// Mitsubishi GX Works2 project: BookEX6_25 Transfer   PLC: Q13UDV

// global labels: Global
VAR_GLOBAL
  bVar0 AT M5000 : BOOL;
  abArray0 AT M5010 : ARRAY [0..49] OF BOOL;
  sStr0 AT D5000 : STRING[199];
  sStr1 AT D5100 : STRING[199];
  sStr2 AT D5200 : STRING[199];
  sStr3 AT D5300 : STRING[199];
  sStr4 AT D5400 : STRING[199];
  sStr5 AT D5500 : STRING[199];
  sStr6 AT D5600 : STRING[199];
  sStr7 AT D5700 : STRING[199];
  sStr8 AT D5800 : STRING[199];
  sStr9 AT D5900 : STRING[199];
  iVar0 AT D4500 : INT;
  iVar1 AT D4501 : INT;
  iVar2 AT D4502 : INT;
  iVar3 AT D4503 : INT;
  iVar4 AT D4504 : INT;
  iVar5 AT D4505 : INT;
  iVar6 AT D4506 : INT;
  iVar7 AT D4507 : INT;
  iVar8 AT D4508 : INT;
  iVar9 AT D4509 : INT;
  dVar0 AT D4510 : DINT;
  dVar1 AT D4512 : DINT;
  dVar2 AT D4514 : DINT;
  dVar3 AT D4516 : DINT;
  dVar4 AT D4518 : DINT;
  dVar5 AT D4520 : DINT;
  dVar6 AT D4522 : DINT;
  dVar7 AT D4524 : DINT;
  dVar8 AT D4526 : DINT;
  dVar9 AT D4528 : DINT;
  wVar0 AT D4530 : WORD;
  wVar1 AT D4531 : WORD;
  wVar2 AT D4532 : WORD;
  wVar3 AT D4533 : WORD;
  wVar4 AT D4534 : WORD;
  wVar5 AT D4535 : WORD;
  wVar6 AT D4536 : WORD;
  wVar7 AT D4537 : WORD;
  wVar8 AT D4538 : WORD;
  wVar9 AT D4539 : WORD;
  dwVar0 AT D4540 : DWORD;
  dwVar1 AT D4542 : DWORD;
  dwVar2 AT D4544 : DWORD;
  dwVar3 AT D4546 : DWORD;
  dwVar4 AT D4548 : DWORD;
  dwVar5 AT D4550 : DWORD;
  dwVar6 AT D4552 : DWORD;
  dwVar7 AT D4554 : DWORD;
  dwVar8 AT D4556 : DWORD;
  dwVar9 AT D4558 : DWORD;
  fsVar0 AT D4560 : REAL;
  fsVar1 AT D4562 : REAL;
  fsVar2 AT D4564 : REAL;
  fsVar3 AT D4566 : REAL;
  fsVar4 AT D4568 : REAL;
  fsVar5 AT D4570 : REAL;
  fsVar6 AT D4572 : REAL;
  fsVar7 AT D4574 : REAL;
  fsVar8 AT D4576 : REAL;
  fsVar9 AT D4578 : REAL;
  fdVar0 AT D4580 : LREAL;
  tTime0 AT D4620 : TIME;
  tTime1 AT D4622 : TIME;
  tTime2 AT D4624 : TIME;
  tTime3 AT D4626 : TIME;
  tTime4 AT D4628 : TIME;
  tTime5 AT D4630 : TIME;
  tTime6 AT D4632 : TIME;
  tTime7 AT D4634 : TIME;
  tTime8 AT D4636 : TIME;
  tTime9 AT D4638 : TIME;
  tTime10 AT D4640 : TIME;
  bVar1 AT M5001 : BOOL;
  bVar2 AT M5002 : BOOL;
  bVar3 AT M5003 : BOOL;
  bVar4 AT M5004 : BOOL;
  bVar5 AT M5005 : BOOL;
  bVar6 AT M5006 : BOOL;
  bVar7 AT M5007 : BOOL;
  bVar8 AT M5008 : BOOL;
  bVar9 AT M5009 : BOOL;
  abArray1 AT M5060 : ARRAY [0..49] OF BOOL;
  abArray2 AT M5110 : ARRAY [0..49] OF BOOL;
  abArray3 AT M5160 : ARRAY [0..49] OF BOOL;
  abArray4 AT M5210 : ARRAY [0..49] OF BOOL;
  abArray5 AT M5260 : ARRAY [0..49] OF BOOL;
  abArray6 AT M5310 : ARRAY [0..49] OF BOOL;
  abArray7 AT M5360 : ARRAY [0..49] OF BOOL;
  abArray8 AT M5410 : ARRAY [0..49] OF BOOL;
  abArray9 AT M5460 : ARRAY [0..49] OF BOOL;
  fdVar1 AT D4584 : LREAL;
  fdVar2 AT D4588 : LREAL;
  fdVar3 AT D4592 : LREAL;
  fdVar4 AT D4596 : LREAL;
  fdVar5 AT D4600 : LREAL;
  fdVar6 AT D4604 : LREAL;
  fdVar7 AT D4608 : LREAL;
  fdVar8 AT D4612 : LREAL;
  fdVar9 AT D4616 : LREAL;
  afsPen0 AT D2000 : ARRAY [0..499] OF REAL;
  afsPen1 AT D3000 : ARRAY [0..499] OF REAL;
  adwD10 AT D10 : ARRAY [0..9] OF DWORD;
  awD10 AT D10 : ARRAY [0..19] OF WORD;
  abM10 AT M10 : ARRAY [0..7] OF BOOL;
END_VAR
// user libraries (not included): HMI

PROGRAM ExBMOV
VAR
  Mov4WORD_1 : Mov4WORD;
  Mov4WORD_2 : Mov4WORD;
  Mov4WORD_3 : Mov4WORD;
  Mov4WORD_4 : Mov4WORD;
  Mov8INT_1 : Mov8INT;
  Mov4WORD_5 : Mov4WORD;
  aMacNo1 : ARRAY [0..9] OF INT;
  aMacNo2 : ARRAY [0..9] OF INT;
  aMacNo3 : ARRAY [0..9] OF INT;
  aMacNo4 : ARRAY [0..9] OF INT;
END_VAR
(* structured ladder/FBD written out as ST: instructions are called as NAME(EN, inputs, outputs); _pN, _eN, _tN stand for wires *)
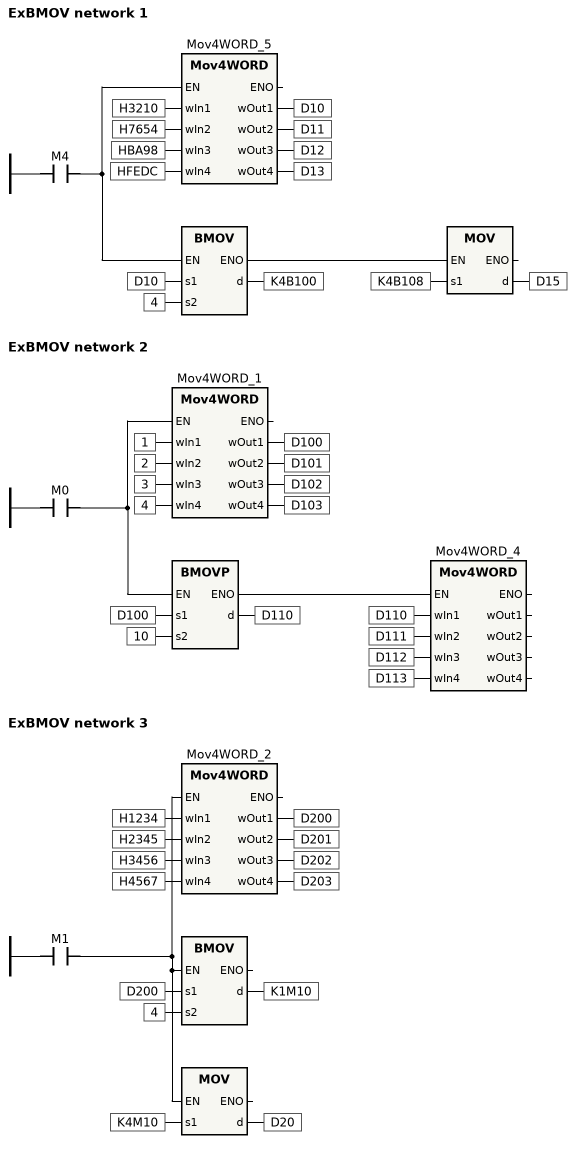
(* network 1 *)
Mov4WORD_5(EN := M4, wIn1 := H3210, wIn2 := H7654, wIn3 := HBA98, wIn4 := HFEDC, wOut1 => D10, wOut2 => D11, wOut3 => D12, wOut4 => D13);
_e1 := BMOV(M4, D10, 4, K4B100);
MOV(_e1, K4B108, D15);
(* network 2 *)
Mov4WORD_1(EN := M0, wIn1 := 1, wIn2 := 2, wIn3 := 3, wIn4 := 4, wOut1 => D100, wOut2 => D101, wOut3 => D102, wOut4 => D103);
_e1 := BMOVP(M0, D100, 10, D110);
Mov4WORD_4(EN := _e1, wIn1 := D110, wIn2 := D111, wIn3 := D112, wIn4 := D113);
(* network 3 *)
Mov4WORD_2(EN := M1, wIn1 := H1234, wIn2 := H2345, wIn3 := H3456, wIn4 := H4567, wOut1 => D200, wOut2 => D201, wOut3 => D202, wOut4 => D203);
BMOV(M1, D200, 4, K1M10);
MOV(M1, K4M10, D20);
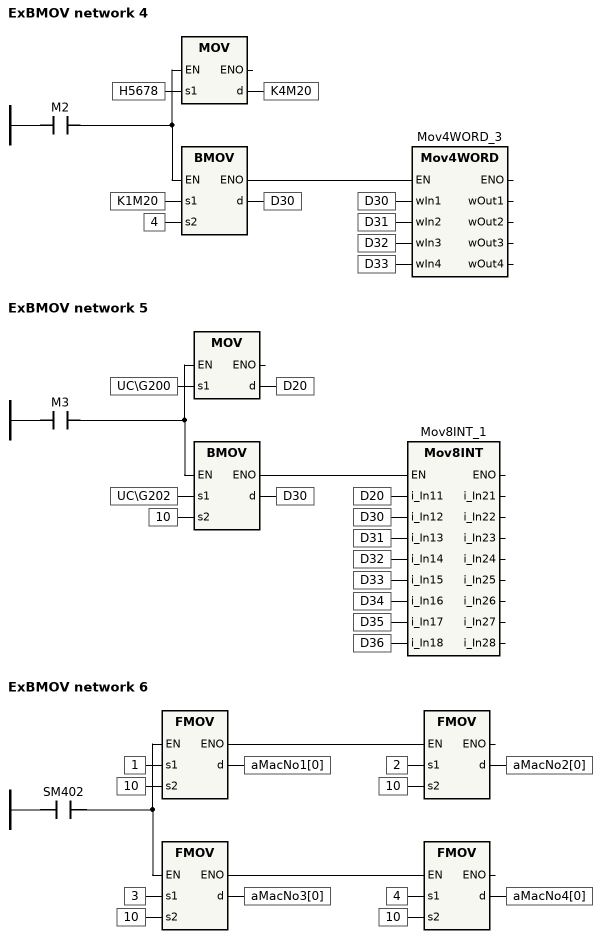
(* network 4 *)
MOV(M2, H5678, K4M20);
_e1 := BMOV(M2, K1M20, 4, D30);
Mov4WORD_3(EN := _e1, wIn1 := D30, wIn2 := D31, wIn3 := D32, wIn4 := D33);
(* network 5 *)
MOV(M3, UC\G200, D20);
_e1 := BMOV(M3, UC\G202, 10, D30);
Mov8INT_1(EN := _e1, i_In11 := D20, i_In12 := D30, i_In13 := D31, i_In14 := D32, i_In15 := D33, i_In16 := D34, i_In17 := D35, i_In18 := D36);
(* network 6 *)
_e1 := FMOV(SM402, 1, 10, aMacNo1[0]);
FMOV(_e1, 2, 10, aMacNo2[0]);
_e2 := FMOV(SM402, 3, 10, aMacNo3[0]);
FMOV(_e2, 4, 10, aMacNo4[0]);
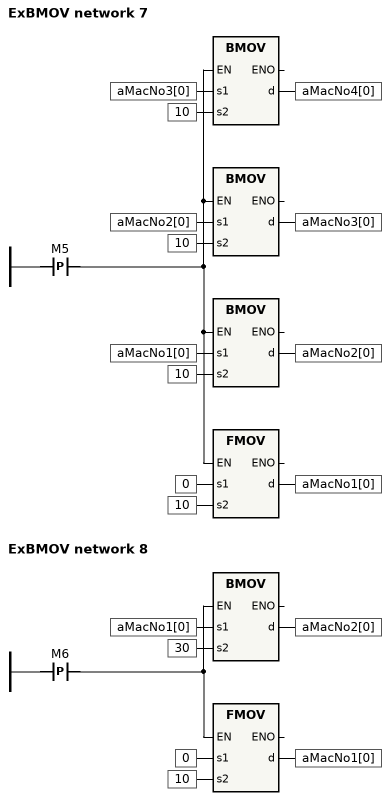
(* network 7 *)
_p1 := LDP(TRUE, M5);
BMOV(_p1, aMacNo3[0], 10, aMacNo4[0]);
BMOV(_p1, aMacNo2[0], 10, aMacNo3[0]);
BMOV(_p1, aMacNo1[0], 10, aMacNo2[0]);
FMOV(_p1, 0, 10, aMacNo1[0]);
(* network 8 *)
_p1 := LDP(TRUE, M6);
BMOV(_p1, aMacNo1[0], 30, aMacNo2[0]);
FMOV(_p1, 0, 10, aMacNo1[0]);
END_PROGRAM

PROGRAM ExCML
VAR
  HMI20_1 : HMI20;
END_VAR
(* structured ladder/FBD written out as ST: instructions are called as NAME(EN, inputs, outputs); _pN, _eN, _tN stand for wires *)
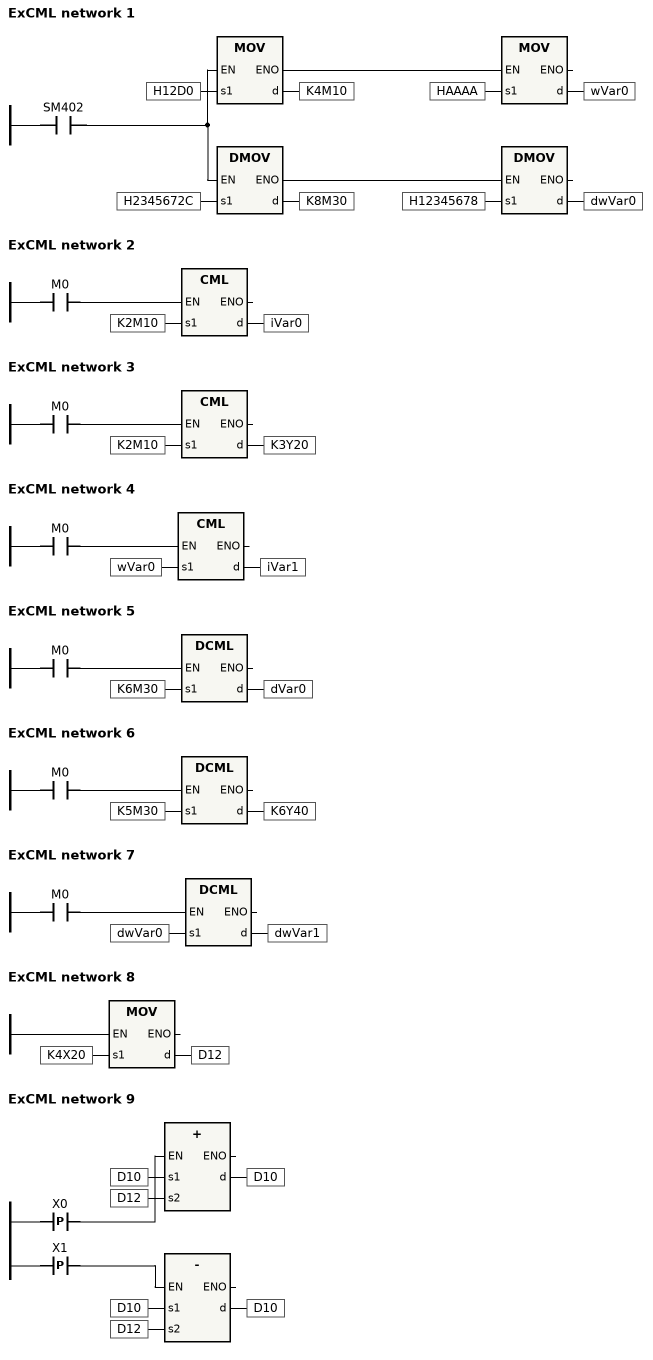
(* network 1 *)
_e1 := MOV(SM402, H12D0, K4M10);
MOV(_e1, HAAAA, wVar0);
_e2 := DMOV(SM402, H2345672C, K8M30);
DMOV(_e2, H12345678, dwVar0);
(* network 2 *)
CML(M0, K2M10, iVar0);
(* network 3 *)
CML(M0, K2M10, K3Y20);
(* network 4 *)
CML(M0, wVar0, iVar1);
(* network 5 *)
DCML(M0, K6M30, dVar0);
(* network 6 *)
DCML(M0, K5M30, K6Y40);
(* network 7 *)
DCML(M0, dwVar0, dwVar1);
(* network 8 *)
MOV(TRUE, K4X20, D12);
(* network 9 *)
+(LDP(TRUE, X0), D10, D12, D10);
-(LDP(TRUE, X1), D10, D12, D10);
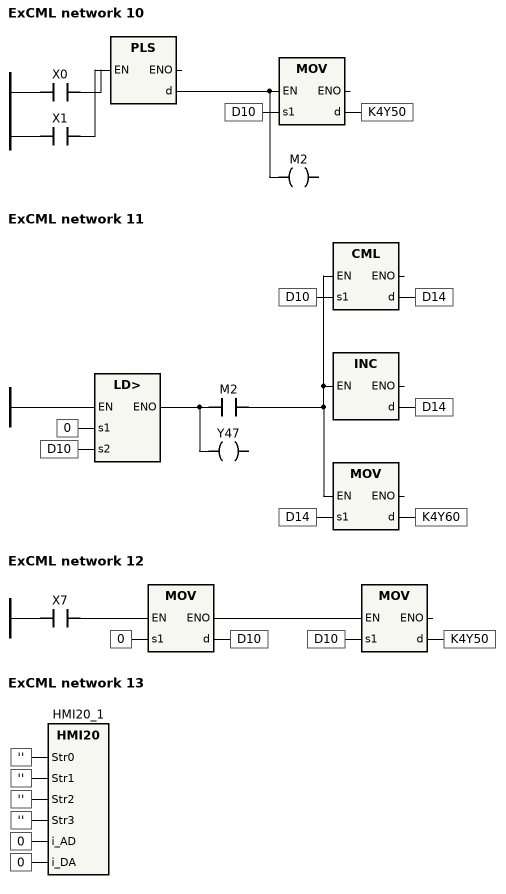
(* network 10 *)
PLS(X0 OR X1, _t1);
M2 := _t1;
MOV(_t1, D10, K4Y50);
(* network 11 *)
_e1 := LD>(TRUE, 0, D10);
_p2 := _e1 AND M2;
CML(_p2, D10, D14);
INC(_p2, D14);
MOV(_p2, D14, K4Y60);
Y47 := _e1;
(* network 12 *)
_e1 := MOV(X7, 0, D10);
MOV(_e1, D10, K4Y50);
(* network 13 *)
HMI20_1(Str0 := '', Str1 := '', Str2 := '', Str3 := '', i_AD := 0, i_DA := 0);
END_PROGRAM

PROGRAM ExFMOV
VAR
  Mov4WORD_1 : Mov4WORD;
  Mov4WORD_2 : Mov4WORD;
  Mov4WORD_3 : Mov4WORD;
  Mov4WORD_4 : Mov4WORD;
  Mov4DWORD_1 : Mov4DWORD;
  aiData : ARRAY [0..9] OF INT;
  adwData : ARRAY [0..9] OF DWORD;
  HMI20_1 : HMI20;
END_VAR
(* structured ladder/FBD written out as ST: instructions are called as NAME(EN, inputs, outputs); _pN, _eN, _tN stand for wires *)
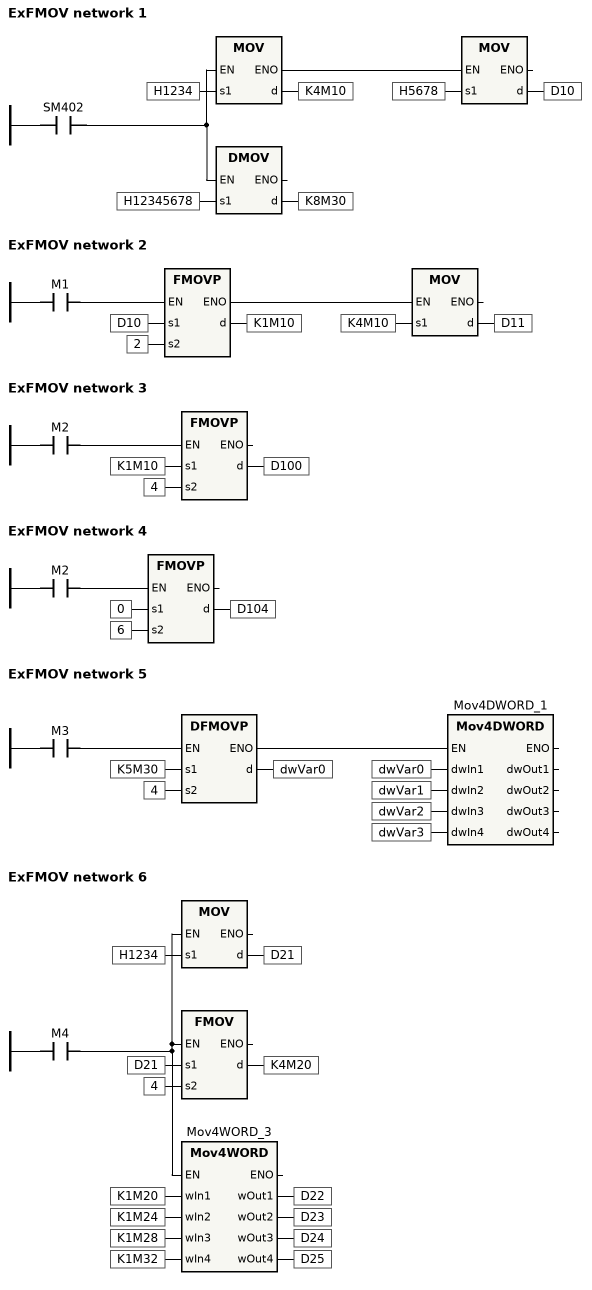
(* network 1 *)
_e1 := MOV(SM402, H1234, K4M10);
MOV(_e1, H5678, D10);
DMOV(SM402, H12345678, K8M30);
(* network 2 *)
_e1 := FMOVP(M1, D10, 2, K1M10);
MOV(_e1, K4M10, D11);
(* network 3 *)
FMOVP(M2, K1M10, 4, D100);
(* network 4 *)
FMOVP(M2, 0, 6, D104);
(* network 5 *)
_e1 := DFMOVP(M3, K5M30, 4, dwVar0);
Mov4DWORD_1(EN := _e1, dwIn1 := dwVar0, dwIn2 := dwVar1, dwIn3 := dwVar2, dwIn4 := dwVar3);
(* network 6 *)
MOV(M4, H1234, D21);
FMOV(M4, D21, 4, K4M20);
Mov4WORD_3(EN := M4, wIn1 := K1M20, wIn2 := K1M24, wIn3 := K1M28, wIn4 := K1M32, wOut1 => D22, wOut2 => D23, wOut3 => D24, wOut4 => D25);
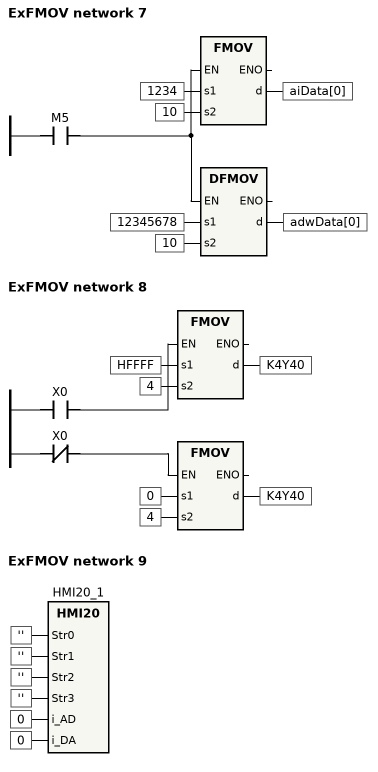
(* network 7 *)
FMOV(M5, 1234, 10, aiData[0]);
DFMOV(M5, 12345678, 10, adwData[0]);
(* network 8 *)
FMOV(X0, HFFFF, 4, K4Y40);
FMOV(NOT X0, 0, 4, K4Y40);
(* network 9 *)
HMI20_1(Str0 := '', Str1 := '', Str2 := '', Str3 := '', i_AD := 0, i_DA := 0);
END_PROGRAM

PROGRAM ExMOV
VAR
  Mov4WORD_1 : Mov4WORD;
END_VAR
(* structured ladder/FBD written out as ST: instructions are called as NAME(EN, inputs, outputs); _pN, _eN, _tN stand for wires *)
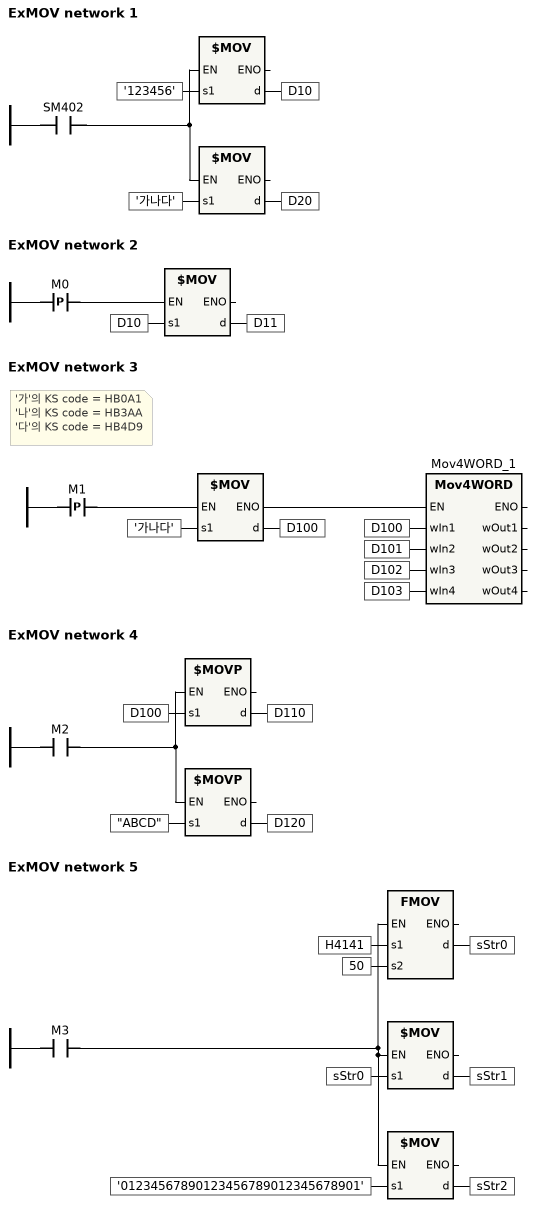
(* network 1 *)
$MOV(SM402, '123456', D10);
$MOV(SM402, '가나다', D20);
(* network 2 *)
$MOV(LDP(TRUE, M0), D10, D11);
(* network 3 *)
(* '가'의 KS code = HB0A1 / '나'의 KS code = HB3AA / '다'의 KS code = HB4D9 *)
_e1 := $MOV(LDP(TRUE, M1), '가나다', D100);
Mov4WORD_1(EN := _e1, wIn1 := D100, wIn2 := D101, wIn3 := D102, wIn4 := D103);
(* network 4 *)
$MOVP(M2, D100, D110);
$MOVP(M2, "ABCD", D120);
(* network 5 *)
FMOV(M3, H4141, 50, sStr0);
$MOV(M3, sStr0, sStr1);
$MOV(M3, '01234567890123456789012345678901', sStr2);
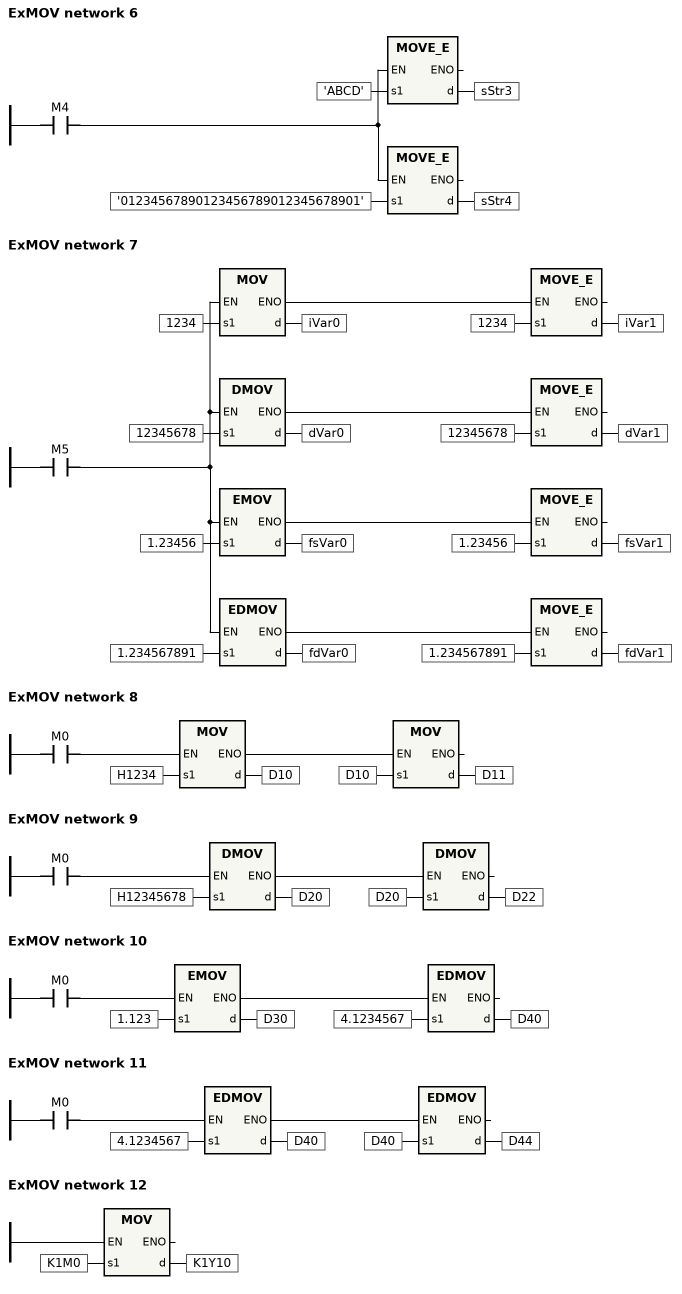
(* network 6 *)
MOVE_E(M4, 'ABCD', sStr3);
MOVE_E(M4, '01234567890123456789012345678901', sStr4);
(* network 7 *)
_e1 := MOV(M5, 1234, iVar0);
MOVE_E(_e1, 1234, iVar1);
_e2 := DMOV(M5, 12345678, dVar0);
MOVE_E(_e2, 12345678, dVar1);
_e3 := EMOV(M5, 1.23456, fsVar0);
MOVE_E(_e3, 1.23456, fsVar1);
_e4 := EDMOV(M5, 1.234567891, fdVar0);
MOVE_E(_e4, 1.234567891, fdVar1);
(* network 8 *)
_e1 := MOV(M0, H1234, D10);
MOV(_e1, D10, D11);
(* network 9 *)
_e1 := DMOV(M0, H12345678, D20);
DMOV(_e1, D20, D22);
(* network 10 *)
_e1 := EMOV(M0, 1.123, D30);
EDMOV(_e1, 4.1234567, D40);
(* network 11 *)
_e1 := EDMOV(M0, 4.1234567, D40);
EDMOV(_e1, D40, D44);
(* network 12 *)
MOV(TRUE, K1M0, K1Y10);
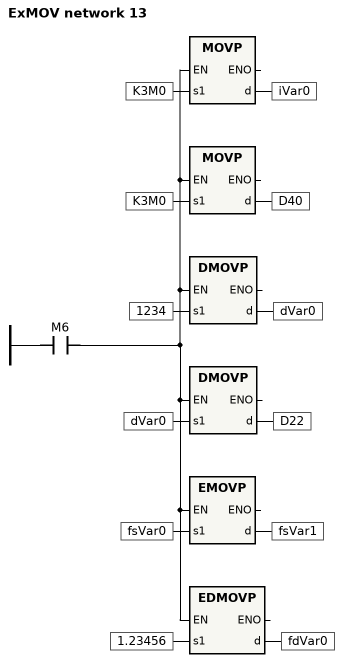
(* network 13 *)
MOVP(M6, K3M0, iVar0);
MOVP(M6, K3M0, D40);
DMOVP(M6, 1234, dVar0);
DMOVP(M6, dVar0, D22);
EMOVP(M6, fsVar0, fsVar1);
EDMOVP(M6, 1.23456, fdVar0);
END_PROGRAM

PROGRAM ExSWAP
VAR
  Mov8INT_1 : Mov8INT;
  Mov8INT_2 : Mov8INT;
  Mov8INT_3 : Mov8INT;
  Mov8INT_4 : Mov8INT;
  BSWAP_1 : BSWAP;
END_VAR
(* structured ladder/FBD written out as ST: instructions are called as NAME(EN, inputs, outputs); _pN, _eN, _tN stand for wires *)
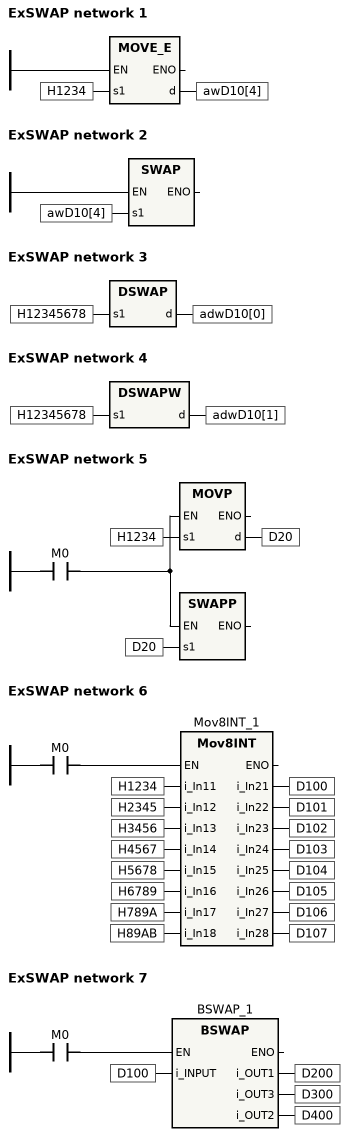
(* network 1 *)
MOVE_E(TRUE, H1234, awD10[4]);
(* network 2 *)
SWAP(TRUE, awD10[4]);
(* network 3 *)
adwD10[0] := DSWAP(H12345678);
(* network 4 *)
adwD10[1] := DSWAPW(H12345678);
(* network 5 *)
MOVP(M0, H1234, D20);
SWAPP(M0, D20);
(* network 6 *)
Mov8INT_1(EN := M0, i_In11 := H1234, i_In12 := H2345, i_In13 := H3456, i_In14 := H4567, i_In15 := H5678, i_In16 := H6789, i_In17 := H789A, i_In18 := H89AB, i_In21 => D100, i_In22 => D101, i_In23 => D102, i_In24 => D103, i_In25 => D104, i_In26 => D105, i_In27 => D106, i_In28 => D107);
(* network 7 *)
BSWAP_1(EN := M0, i_INPUT := D100, i_OUT1 => D200, i_OUT3 => D300, i_OUT2 => D400);
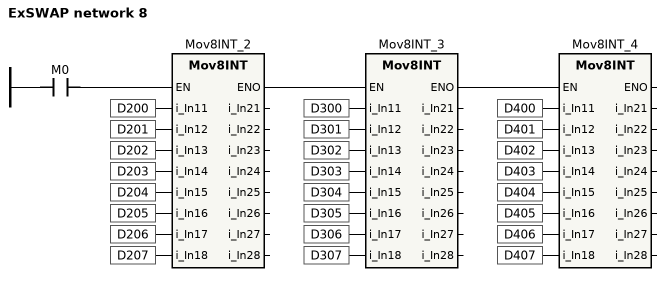
(* network 8 *)
Mov8INT_2(EN := M0, i_In11 := D200, i_In12 := D201, i_In13 := D202, i_In14 := D203, i_In15 := D204, i_In16 := D205, i_In17 := D206, i_In18 := D207);
Mov8INT_3(EN := Mov8INT_2.ENO, i_In11 := D300, i_In12 := D301, i_In13 := D302, i_In14 := D303, i_In15 := D304, i_In16 := D305, i_In17 := D306, i_In18 := D307);
Mov8INT_4(EN := Mov8INT_3.ENO, i_In11 := D400, i_In12 := D401, i_In13 := D402, i_In14 := D403, i_In15 := D404, i_In16 := D405, i_In17 := D406, i_In18 := D407);
END_PROGRAM

PROGRAM ExXCH
VAR
  Mov4INT_1 : Mov4INT;
  Mov4INT_2 : Mov4INT;
END_VAR
(* structured ladder/FBD written out as ST: instructions are called as NAME(EN, inputs, outputs); _pN, _eN, _tN stand for wires *)
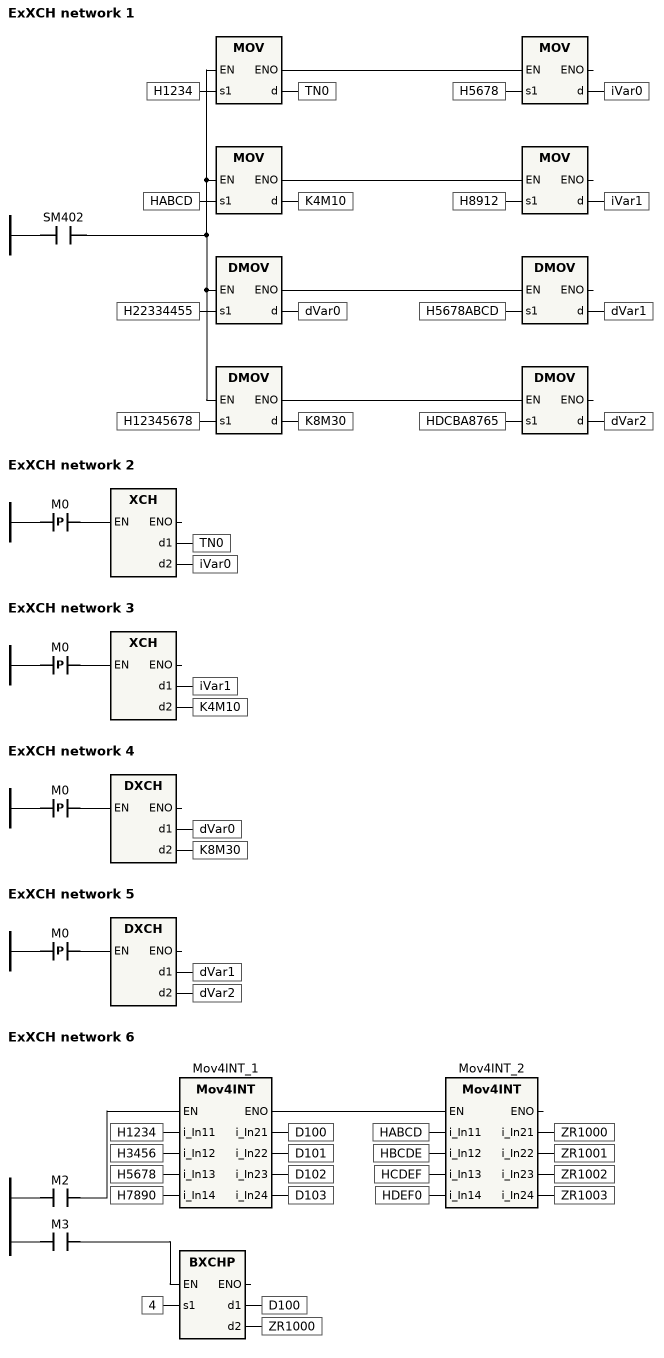
(* network 1 *)
_e1 := MOV(SM402, H1234, TN0);
MOV(_e1, H5678, iVar0);
_e2 := MOV(SM402, HABCD, K4M10);
MOV(_e2, H8912, iVar1);
_e3 := DMOV(SM402, H22334455, dVar0);
DMOV(_e3, H5678ABCD, dVar1);
_e4 := DMOV(SM402, H12345678, K8M30);
DMOV(_e4, HDCBA8765, dVar2);
(* network 2 *)
XCH(LDP(TRUE, M0), TN0, iVar0);
(* network 3 *)
XCH(LDP(TRUE, M0), iVar1, K4M10);
(* network 4 *)
DXCH(LDP(TRUE, M0), dVar0, K8M30);
(* network 5 *)
DXCH(LDP(TRUE, M0), dVar1, dVar2);
(* network 6 *)
Mov4INT_1(EN := M2, i_In11 := H1234, i_In12 := H3456, i_In13 := H5678, i_In14 := H7890, i_In21 => D100, i_In22 => D101, i_In23 => D102, i_In24 => D103);
Mov4INT_2(EN := Mov4INT_1.ENO, i_In11 := HABCD, i_In12 := HBCDE, i_In13 := HCDEF, i_In14 := HDEF0, i_In21 => ZR1000, i_In22 => ZR1001, i_In23 => ZR1002, i_In24 => ZR1003);
BXCHP(M3, 4, D100, ZR1000);
END_PROGRAM

FUNCTION DSWAP
VAR_INPUT
  i_DW : DWORD;
END_VAR
VAR
  wLow : WORD;
  wHigh : WORD;
  dwLow : DWORD;
  dwHigh : DWORD;
END_VAR
;
wLow := DWORD_TO_WORD(i_DW);
wHigh := DWORD_TO_WORD(SHR(i_DW,16));
SWAP(TRUE, wLow);
SWAP(TRUE, wHigh);
dwLow := WORD_TO_DWORD(wLow);
dwHigh := SHL(WORD_TO_DWORD(wHigh), 16);
DSWAP := dwHigh OR dwLow;
END_FUNCTION

FUNCTION DSWAPW
VAR_INPUT
  i_DW : DWORD;
END_VAR
VAR
  dwLow : DWORD;
  dwHigh : DWORD;
END_VAR
;
dwHigh := SHR(i_DW,16); 
dwLow := SHL(i_DW, 16);
DSWAPW := dwHigh OR dwLow;
END_FUNCTION

FUNCTION_BLOCK BSWAP
VAR_INPUT
  i_INPUT : INT;
END_VAR
VAR_OUTPUT
  i_OUT1 : INT;
  i_OUT3 : INT;
  i_OUT2 : INT;
END_VAR
VAR
  Buffer : ARRAY [0..98] OF INT;
  ix : INT;
  Buffer2 : ARRAY [0..98] OF INT;
END_VAR
;

BMOV(TRUE, i_INPUT, 8, Buffer[0]); 
BMOV(TRUE, i_INPUT, 8, Buffer2[0]); 
BMOV(TRUE, Buffer[0], 8, i_OUT1); 
FOR ix := 0 TO 7 DO 
	SWAP(TRUE, Buffer[ix]);	 
END_FOR;
BMOV(TRUE, Buffer[0], 8, i_OUT2); 
FOR ix := 0 TO 3 DO 
	XCH(TRUE, Buffer2[7-ix], Buffer2[ix]); 
END_FOR;
BMOV(TRUE, Buffer2[0], 8, i_OUT3);
END_FUNCTION_BLOCK
